ABB RAPID module: Module1.mod

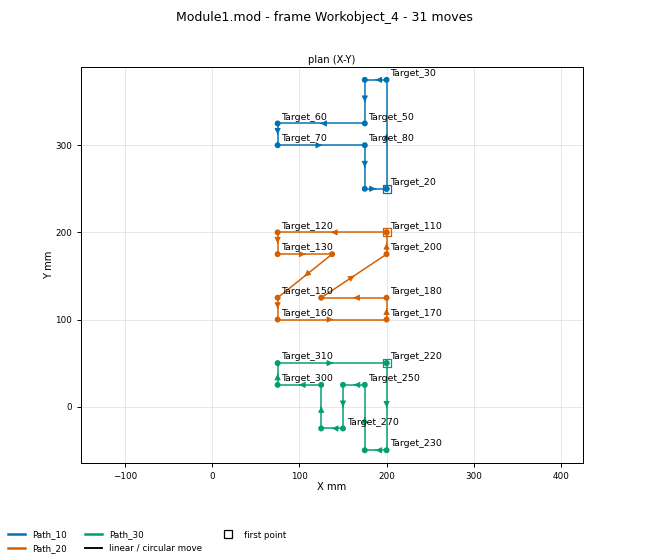
[picture p0: tool path of Module1.mod in frame Workobject_4, 31 of 34 moves have a stored position in this frame; points joined in program order, loops and branches not executed]
MODULE Module1
        CONST robtarget Target_20:=[[200,250,0],[0,0,1,0],[0,0,0,0],[9E+09,9E+09,9E+09,9E+09,9E+09,9E+09]];
    CONST robtarget Target_30:=[[200,375,0],[0,0,1,0],[0,0,0,0],[9E+09,9E+09,9E+09,9E+09,9E+09,9E+09]];
    CONST robtarget Target_40:=[[175,375,0],[0,0,1,0],[0,0,0,0],[9E+09,9E+09,9E+09,9E+09,9E+09,9E+09]];
    CONST robtarget Target_50:=[[175,325,0],[0,0,1,0],[0,0,0,0],[9E+09,9E+09,9E+09,9E+09,9E+09,9E+09]];
    CONST robtarget Target_60:=[[75,325,0],[0,0,1,0],[0,0,0,0],[9E+09,9E+09,9E+09,9E+09,9E+09,9E+09]];
    CONST robtarget Target_70:=[[75,300,0],[0,0,1,0],[0,0,0,0],[9E+09,9E+09,9E+09,9E+09,9E+09,9E+09]];
    CONST robtarget Target_80:=[[175,300,0],[0,0,1,0],[0,0,0,0],[9E+09,9E+09,9E+09,9E+09,9E+09,9E+09]];
    CONST robtarget Target_90:=[[175,250,0],[0,0,1,0],[0,0,0,0],[9E+09,9E+09,9E+09,9E+09,9E+09,9E+09]];
    CONST robtarget Target_100:=[[200,250,0],[0,0,1,0],[0,0,0,0],[9E+09,9E+09,9E+09,9E+09,9E+09,9E+09]];
    CONST robtarget Target_110:=[[200,200,0],[0,0,1,0],[0,0,0,0],[9E+09,9E+09,9E+09,9E+09,9E+09,9E+09]];
    CONST robtarget Target_120:=[[75,200,0],[0,0,1,0],[0,0,0,0],[9E+09,9E+09,9E+09,9E+09,9E+09,9E+09]];
    CONST robtarget Target_130:=[[75,175,0],[0,0,1,0],[0,0,0,0],[9E+09,9E+09,9E+09,9E+09,9E+09,9E+09]];
    CONST robtarget Target_140:=[[137.5,175,0],[0,0,1,0],[0,0,0,0],[9E+09,9E+09,9E+09,9E+09,9E+09,9E+09]];
    CONST robtarget Target_150:=[[75,125,0],[0,0,1,0],[0,0,0,0],[9E+09,9E+09,9E+09,9E+09,9E+09,9E+09]];
    CONST robtarget Target_160:=[[75,100,0],[0,0,1,0],[0,0,0,0],[9E+09,9E+09,9E+09,9E+09,9E+09,9E+09]];
    CONST robtarget Target_170:=[[200,100,0],[0,0,1,0],[0,0,0,0],[9E+09,9E+09,9E+09,9E+09,9E+09,9E+09]];
    CONST robtarget Target_180:=[[200,125,0],[0,0,1,0],[0,0,0,0],[9E+09,9E+09,9E+09,9E+09,9E+09,9E+09]];
    CONST robtarget Target_190:=[[125,125,0],[0,0,1,0],[0,0,0,0],[9E+09,9E+09,9E+09,9E+09,9E+09,9E+09]];
    CONST robtarget Target_200:=[[200,175,0],[0,0,1,0],[0,0,0,0],[9E+09,9E+09,9E+09,9E+09,9E+09,9E+09]];
    CONST robtarget Target_210:=[[200,200,0],[0,0,1,0],[0,0,0,0],[9E+09,9E+09,9E+09,9E+09,9E+09,9E+09]];
    CONST robtarget Target_220:=[[200,50,0],[0,0,1,0],[0,0,0,0],[9E+09,9E+09,9E+09,9E+09,9E+09,9E+09]];
    CONST robtarget Target_230:=[[200,-50,0],[0,0,1,0],[-1,0,-1,0],[9E+09,9E+09,9E+09,9E+09,9E+09,9E+09]];
    CONST robtarget Target_240:=[[175,-50,0],[0,0,1,0],[-1,0,-1,0],[9E+09,9E+09,9E+09,9E+09,9E+09,9E+09]];
    CONST robtarget Target_250:=[[175,25,0],[0,0,1,0],[0,0,0,0],[9E+09,9E+09,9E+09,9E+09,9E+09,9E+09]];
    CONST robtarget Target_260:=[[150,25,0],[0,0,1,0],[0,0,0,0],[9E+09,9E+09,9E+09,9E+09,9E+09,9E+09]];
    CONST robtarget Target_270:=[[150,-25,0],[0,0,1,0],[-1,0,-1,0],[9E+09,9E+09,9E+09,9E+09,9E+09,9E+09]];
    CONST robtarget Target_280:=[[125,-25,0],[0,0,1,0],[-1,0,-1,0],[9E+09,9E+09,9E+09,9E+09,9E+09,9E+09]];
    CONST robtarget Target_290:=[[125,25,0],[0,0,1,0],[0,0,0,0],[9E+09,9E+09,9E+09,9E+09,9E+09,9E+09]];
    CONST robtarget Target_300:=[[75,25,0],[0,0,1,0],[0,0,0,0],[9E+09,9E+09,9E+09,9E+09,9E+09,9E+09]];
    CONST robtarget Target_310:=[[75,50,0],[0,0,1,0],[0,0,0,0],[9E+09,9E+09,9E+09,9E+09,9E+09,9E+09]];
    CONST robtarget Target_320:=[[200,50,0],[0,0,1,0],[0,0,0,0],[9E+09,9E+09,9E+09,9E+09,9E+09,9E+09]];
    CONST jointtarget JointTarget_1:=[[0,0,0,0,0,0],[9E+09,9E+09,9E+09,9E+09,9E+09,9E+09]];
    CONST jointtarget JointTarget_6:=[[20,30,25,30,15,0],[9E+09,9E+09,9E+09,9E+09,9E+09,9E+09]];
    CONST jointtarget JointTarget_7:=[[90,0,0,0,0,0],[9E+09,9E+09,9E+09,9E+09,9E+09,9E+09]];
!***********************************************************
    !
    ! Módulo:  Module1
    !
    ! Descripción:
    !   <Introduzca la descripción aquí>
    !
    ! Autor: ASUS
    !
    ! Versión: 1.0
    !
    !***********************************************************


    !***********************************************************
    !
    ! Procedimiento Main
    !
    !   Este es el punto de entrada de su programa
    !
    !***********************************************************
    PROC main()
        !Añada aquí su código
        WaitDI DI_01,1;
        SetDO DO_03,1;
        Path_40;
        Path_50;
        Path_10;
        Path_50;
        Path_20;
        Path_50;
        Path_30;
        Path_50;
        Path_40;
        WaitDI DI_02,1;
        Path_60;
        SetDO DO_03,0;

    ENDPROC
    PROC Path_10()
        MoveL Target_20,v100,z1,MyNewTool\WObj:=Workobject_4;
        MoveL Target_30,v100,z1,MyNewTool\WObj:=Workobject_4;
        MoveL Target_40,v100,z1,MyNewTool\WObj:=Workobject_4;
        MoveL Target_50,v100,z1,MyNewTool\WObj:=Workobject_4;
        MoveL Target_60,v100,z1,MyNewTool\WObj:=Workobject_4;
        MoveL Target_70,v100,z1,MyNewTool\WObj:=Workobject_4;
        MoveL Target_80,v100,z1,MyNewTool\WObj:=Workobject_4;
        MoveL Target_90,v100,z1,MyNewTool\WObj:=Workobject_4;
        MoveL Target_100,v100,z1,MyNewTool\WObj:=Workobject_4;
    ENDPROC
    PROC Path_20()
        MoveL Target_110,v100,z1,MyNewTool\WObj:=Workobject_4;
        MoveL Target_120,v100,z1,MyNewTool\WObj:=Workobject_4;
        MoveL Target_130,v100,z1,MyNewTool\WObj:=Workobject_4;
        MoveL Target_140,v100,z1,MyNewTool\WObj:=Workobject_4;
        MoveL Target_150,v100,z1,MyNewTool\WObj:=Workobject_4;
        MoveL Target_160,v100,z1,MyNewTool\WObj:=Workobject_4;
        MoveL Target_170,v100,z1,MyNewTool\WObj:=Workobject_4;
        MoveL Target_180,v100,z1,MyNewTool\WObj:=Workobject_4;
        MoveL Target_190,v100,z1,MyNewTool\WObj:=Workobject_4;
        MoveL Target_200,v100,z1,MyNewTool\WObj:=Workobject_4;
        MoveL Target_210,v100,z1,MyNewTool\WObj:=Workobject_4;
    ENDPROC
    PROC Path_30()
        MoveL Target_220,v100,z1,MyNewTool\WObj:=Workobject_4;
        MoveL Target_230,v100,z1,MyNewTool\WObj:=Workobject_4;
        MoveL Target_240,v100,z1,MyNewTool\WObj:=Workobject_4;
        MoveL Target_250,v100,z1,MyNewTool\WObj:=Workobject_4;
        MoveL Target_260,v100,z1,MyNewTool\WObj:=Workobject_4;
        MoveL Target_270,v100,z1,MyNewTool\WObj:=Workobject_4;
        MoveL Target_280,v100,z1,MyNewTool\WObj:=Workobject_4;
        MoveL Target_290,v100,z1,MyNewTool\WObj:=Workobject_4;
        MoveL Target_300,v100,z1,MyNewTool\WObj:=Workobject_4;
        MoveL Target_310,v100,z1,MyNewTool\WObj:=Workobject_4;
        MoveL Target_320,v100,z1,MyNewTool\WObj:=Workobject_4;
    ENDPROC
    PROC Path_40()
        MoveAbsJ JointTarget_1,v1000,z100,MyNewTool\WObj:=Workobject_4;
    ENDPROC
    PROC Path_50()
        MoveAbsJ JointTarget_6,v1000,z100,MyNewTool\WObj:=Workobject_4;
    ENDPROC
    PROC Path_60()
        MoveAbsJ JointTarget_7,v1000,z100,MyNewTool\WObj:=Workobject_4;
    ENDPROC
ENDMODULE
